TYPE dut_hmi_Analogue :
STRUCT
	Value:REAL;
	Per_thousand:REAL;
	Colour:INT;
END_STRUCT
END_TYPE

(* stored: Version 1.1.0.1, ProductVersion 3.1.4024.0
   DUT dut_hmi_Analogue: Id {2003ebf0-55bc-4c2a-a795-cfd07c1d5fac} *)
